{attribute 'reflection'} 
FUNCTION_BLOCK FB_Sample 
VAR 
    {attribute 'instance-path'} 
    {attribute 'noinit'} 
    sPath : STRING; 
END_VAR

END_FUNCTION_BLOCK

(* stored: Version 1.1.0.1, ProductVersion 3.1.4024.12
   POU FB_Sample: Id {2aa8f178-7ea8-4256-b8d2-7cd95ddd0a8b}, SpecialFunc None *)
